(* PLC project PLC1, Beckhoff Automation GmbH TwinCAT PLC Control 3.5.21.30 *)
(* stored: creationDateTime 2026-05-11T22:43:36.8488113, modificationDateTime 2026-05-11T22:43:36.8527705 *)

FUNCTION F_CreateCPULoad
VAR_INPUT
	nIterations : DINT := 500000; (* Tune this to adjust load *)
END_VAR

VAR
	iIter  : DINT;
	fAccum : LREAL := 0.0;
END_VAR

            FOR iIter := 1 TO nIterations DO
	fAccum := fAccum + SQRT(DINT_TO_LREAL(iIter));
END_FOR
          
END_FUNCTION
